{attribute 'qualified_only'}
{attribute 'strict'}
TYPE E_ViseJawState :
(
	P1_0_120,
	P2_80_210
);
END_TYPE

(* stored: Version 1.1.0.1, ProductVersion 3.1.4024.12
   EnumerationTextList E_ViseJawState: Id {e9c4b87c-46a7-4cbd-90f8-c7893e8d9447} *)
